{attribute 'hide_all_locals'}
FUNCTION_BLOCK DisableGroup EXTENDS TaskBase
VAR_INPUT
END_VAR
VAR_OUTPUT
END_VAR
VAR
	groupDisable			: MC_GroupDisable;
	_caGroup			: ICollisionGroup;
	_disableGroup : BOOL;
	Logger : TcMessage_Ext;
END_VAR

METHOD Abort : BOOL
State := 0;
groupDisable.Execute := FALSE;
Abort := true;
END_METHOD

METHOD Cycle : BOOL
VAR_INPUT
END_VAR
CASE State OF
	0:
		IF _disableGroup THEN
			_Done := FALSE;
			_Error := FALSE;
			_Busy := TRUE;
			groupDisable.Execute := TRUE;
			IF groupDisable.Busy THEN
				_disableGroup := FALSE;
				State := 10;
				Logger.Send(TC_EVENTS.XtsCaGroupEvents.CAGroupDisabling,'');
			END_IF
		END_IF
	
	10:
		IF NOT groupDisable.Busy THEN
			IF groupDisable.Done THEN
				_Done := TRUE;
				Logger.Send(TC_EVENTS.XtsCaGroupEvents.CAGroupDisabled,'');
			ELSIF groupDisable.Error THEN
				_Error := TRUE;
				Logger.Send(TC_EVENTS.XtsCaGroupEvents.CAGroupDisableError,'');
			END_IF
			_Busy := FALSE;
			groupDisable.Execute := false;
			State := 0;
		END_IF
END_CASE


groupDisable(AxesGroup := _caGroup.GroupRef);
END_METHOD

METHOD Execute : BOOL
Execute := _disableGroup := TRUE;
END_METHOD

METHOD FB_init : BOOL
VAR_INPUT
	bInitRetains : BOOL; // if TRUE, the retain variables are initialized (warm start / cold start)
	bInCopyCode : BOOL;  // if TRUE, the instance afterwards gets moved into the copy code (online change)
	CAGroup : ICollisionGroup;
END_VAR
_caGroup := CAGroup;
END_METHOD

END_FUNCTION_BLOCK

(* stored: Version 1.1.0.1, ProductVersion 3.1.4024.12
   POU DisableGroup: Id {e309beac-a8f6-4753-8ed9-d8f37883f7b3}, SpecialFunc None
   Method Abort: Id {471c738d-2cd1-4d5e-b4b6-abdacd440e10}
   Method Cycle: Id {8091e283-75fa-4fa7-b8ef-612c591a9cfd}
   Method Execute: Id {957a3466-1261-44df-92f7-84f5463a1c53}
   Method FB_init: Id {70ba3340-3f18-404c-b96e-e566669fbf07} *)
